DATA_BLOCK "Pilz_fb_DB"
{ S7_Optimized_Access := 'FALSE' }
VERSION : 0.1
NON_RETAIN
"Pilz_fb"

BEGIN

END_DATA_BLOCK

